TYPE "LubrValve_ITF"
VERSION : 0.1
// Block: LubrValve_ITF
   STRUCT
      Sts : Struct
         PumpType : Int;
         Running : Bool;
         Error : Bool;
      END_STRUCT;
      Ctrl : Struct
         RstAlarms : Bool;
         WorkReq : Bool;
      END_STRUCT;
      ValveChain : Struct
         ActualValve : Int;
         MaxValve : Int;
      END_STRUCT;
   END_STRUCT;

END_TYPE
